FUNCTION_BLOCK IlckMotVs (* CAT Function Block Type *)
  (* Standard: 61499-2 *)
  (* Version 0.0, 6/3/2026, Schneider Electric, template *)
  PACKAGE SE.Nereda;
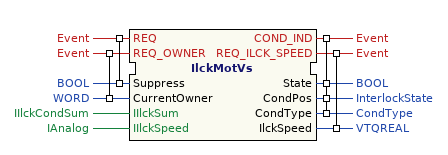
  EVENT_INPUT
    REQ WITH Suppress; (* Request from Socket *)
    REQ_OWNER WITH CurrentOwner;
  END_EVENT
  EVENT_OUTPUT
    COND_IND WITH State, CondPos, CondType; (* Confirmation from Plug *)
    REQ_ILCK_SPEED WITH IlckSpeed; (* Request for new value and limits *)
  END_EVENT
  VAR_INPUT
    Suppress : BOOL; (* 1 = Condition suppressed *)
    CurrentOwner : WORD;
  END_VAR
  VAR_OUTPUT
    State : BOOL; (* 1 = interlock active *)
    CondPos : InterlockState; (* Passive = Passive condition; Active 1 = Active condition 1; Active 2 = Active condition 2 *)
    CondType : CondType; (* Type of condition interlock, (0 = Normal, 1 = Sequential, 2 = Process, 3 = Protection) *)
    IlckSpeed : VTQREAL; (* Vtq value *)
  END_VAR
  SOCKETS
    IIlckSum : IIlckCondSum(DeviceType := BiDirectional, ServiceState := TRUE); (* Interlock condition summary chain input from ilckcondsum block *)
    IIlckSpeed : IAnalog; (* Speed setpoint to be considered if interlock condition is active *)
  END_SOCKETS
  (* Interlock *)
  EVENT_CONNECTIONS
    IIlckSum.CHECK_SERVICE TO IIlckSum.CNF_SERVICE;
    IIlckSum.COND_IND TO COND_IND;
    IIlckSpeed.REQ TO REQ_ILCK_SPEED;
    REQ TO IIlckSum.REQ;
    REQ_OWNER TO IIlckSum.REQ_OWNER;
  END_CONNECTIONS
  DATA_CONNECTIONS
    IIlckSum.State TO State;
    IIlckSum.CondPos TO CondPos;
    IIlckSum.CondType TO CondType;
    IIlckSpeed.Value TO IlckSpeed;
    Suppress TO IIlckSum.Suppress;
    CurrentOwner TO IIlckSum.CurrentOwner;
  END_CONNECTIONS
END_FUNCTION_BLOCK
